// TIA Portal V20 export
VAR_GLOBAL   // PLC tag table "Constantes de Eventos Recibidos"
END_VAR
VAR_GLOBAL CONSTANT   // user constants
   Evento_DISPOSITIVO_PeticionEstadoActual : UInt := 250;
   Evento_DISPOSITIVO_InicioOrdenDipositivo : UInt := 261;
   Evento_DISPOSITIVO_FinalOrdenDispositivo : UInt := 274;
END_VAR
